// TwinCAT 3 PLC project Sample
// ProgramVersion: 3.1.4024.12
// libraries:
//   Tc2_Standard, * (Beckhoff Automation GmbH)
//   Tc2_System, * (Beckhoff Automation GmbH)
//   Tc3_Module, * (Beckhoff Automation GmbH)
// project tree:
//   GVLs/ GVL_Test.TcGVL
//   / PlcTask.TcTTO
//   POUs/ MAIN.TcPOU
// real-time tasks:
//   TASK PlcTask: cycle T#10ms, priority 20, ADS port 350

CONFIGURATION Sample
    RESOURCE PLC ON TwinCAT3
        TASK PlcTask(INTERVAL := T#10ms, PRIORITY := 20);
        PROGRAM MAIN WITH PlcTask : MAIN;
    END_RESOURCE
END_CONFIGURATION

// ---- GVLs/GVL_Test.TcGVL
{attribute 'qualified_only'}
VAR_GLOBAL
	bTestRead: BOOL;	// Bool value to be read by EBC_Measurements
	fTestRead: REAL := -10.0;	// Real value to be read by EBC_Measurements
	
	bTestWrite: BOOL;	// Bool value to be written by EBC_Measurements
	fTestWrite: REAL;	// Real value to be written by EBC_Measurements
	sTestWrite: STRING;	// String value to be written by EBC_Measurements
END_VAR

// ---- POUs/MAIN.TcPOU
PROGRAM MAIN
VAR
	fbTon: Tc2_Standard.TON;
END_VAR

fbTon(IN:=NOT fbTon.Q , PT:=T#1S , Q=> , ET=> );

IF fbTon.Q THEN
	// Update bool
	GVL_Test.bTestRead := NOT GVL_Test.bTestRead;
	// Update real
	IF GVL_Test.fTestRead < 10.0 THEN
		GVL_Test.fTestRead := GVL_Test.fTestRead + 0.5;
	ELSE
		GVL_Test.fTestRead := -10.0;
	END_IF
END_IF

END_PROGRAM
